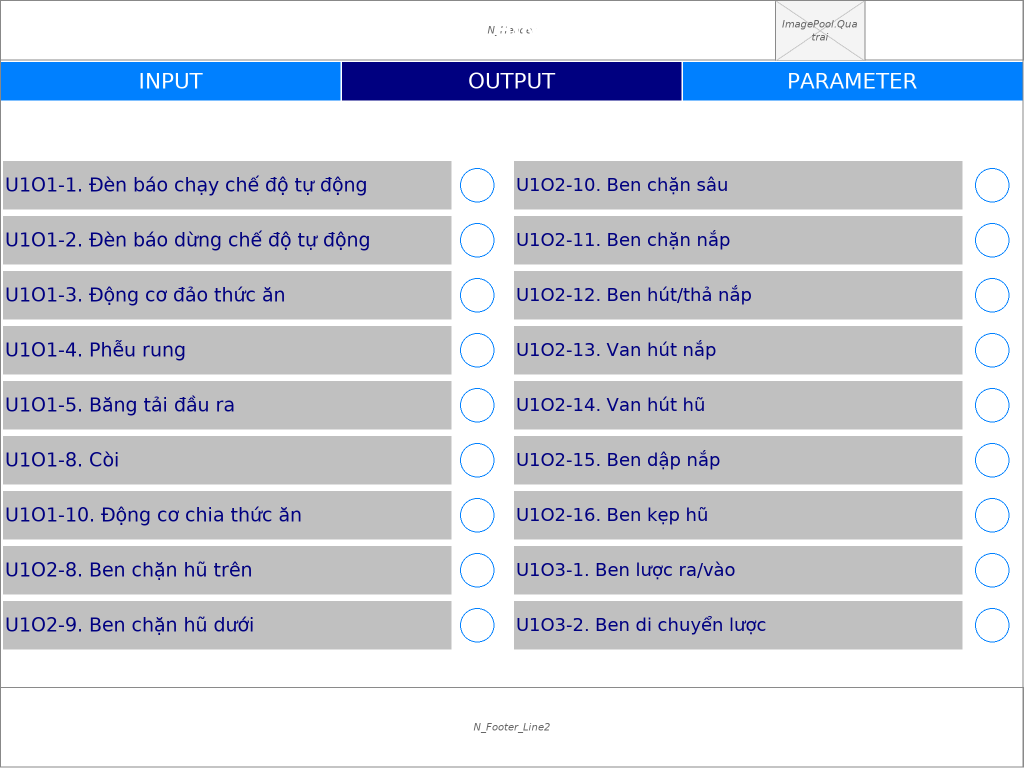
VISUALIZATION N_PLC_O2  // 1024x768
    Frame (0,687 1024x80)
        shows N_Footer_Line2()
    Frame (0,0 1024x60)
        shows N_Header()
    Textfield (353,5 400x50), "MÀN HÌNH IO LINE 2"
    Rectangle (2,160 450x50), "U1O1-1. Đèn báo chạy chế độ tự động"
    Rectangle (2,215 450x50), "U1O1-2. Đèn báo dừng chế độ tự động"
    Rectangle (2,270 450x50), "U1O1-3. Động cơ đảo thức ăn"
    Ellipse (460,168 34x34), colour toggle: GVL_IO.bLight_Running, input disabled if: true
    Ellipse (460,223 34x34), colour toggle: GVL_IO.bLight_Stop, input disabled if: true
    Rectangle (2,325 450x50), "U1O1-4. Phễu rung"
    Rectangle (2,380 450x50), "U1O1-5. Băng tải đầu ra"
    Rectangle (2,435 450x50), "U1O1-8. Còi"
    Rectangle (2,490 450x50), "U1O1-10. Động cơ chia thức ăn"
    Rectangle (2,545 450x50), "U1O2-8. Ben chặn hũ trên"
    Rectangle (2,600 450x50), "U1O2-9. Ben chặn hũ dưới"
    Rectangle (513,160 450x50), "U1O2-10. Ben chặn sâu"
    Rectangle (513,215 450x50), "U1O2-11. Ben chặn nắp"
    Ellipse (460,278 34x34), colour toggle: PR_Line02.fb_FoodMixer.fbInverter.bVFD, input disabled if: true
    Ellipse (460,333 34x34), colour toggle: PR_Line02.fb_WormWeight.fbInverter.bVFD, input disabled if: true
    Ellipse (460,388 34x34), colour toggle: PR_Conveyor_Out.fb_Conveyor.fbInverter.bVFD, input disabled if: true
    Ellipse (460,443 34x34), colour toggle: GVL_IO.bSirens, input disabled if: true
    Ellipse (460,498 34x34), input disabled if: true
    Ellipse (460,553 34x34), colour toggle: PR_Line02.fb_CupSupply.fbCylinder_Up.bMoveExtend, input disabled if: true
    Ellipse (460,608 34x34), colour toggle: PR_Line02.fb_CupSupply.fbCylinder_Dw.bMoveRetract, input disabled if: true
    Ellipse (975,168 34x34), input disabled if: true
    Ellipse (975,223 34x34), colour toggle: PR_Line02.fb_LidSupply.fbCylinder_LidStopper.bMoveRetract, input disabled if: true
    Rectangle (513,270 450x50), "U1O2-12. Ben hút/thả nắp"
    Ellipse (975,278 34x34), input disabled if: true
    Rectangle (513,325 450x50), "U1O2-13. Van hút nắp"
    Rectangle (513,380 450x50), "U1O2-14. Van hút hũ"
    Rectangle (513,435 450x50), "U1O2-15. Ben dập nắp"
    Rectangle (513,490 450x50), "U1O2-16. Ben kẹp hũ"
    Rectangle (513,545 450x50), "U1O3-1. Ben lược ra/vào"
    Rectangle (513,600 450x50), "U1O3-2. Ben di chuyển lược"
    Ellipse (975,333 34x34), input disabled if: true
    Ellipse (975,388 34x34), input disabled if: true
    Ellipse (975,443 34x34), input disabled if: true
    Ellipse (975,498 34x34), colour toggle: PR_Line02.fb_Transfer.fbCylinder_Clip.bMoveRetract, input disabled if: true
    Ellipse (975,553 34x34), colour toggle: PR_Line02.fb_Transfer.fbCylinder_Comb.bMoveExtend, input disabled if: true
    Ellipse (975,608 34x34), colour toggle: PR_Line02.fb_Transfer.fbCylinder_Move_Comb.bMoveExtend, input disabled if: true
    Image (775,0 90x61), image: ImagePool.Qua trai
        OnMouseClick: change screen: N_PLC_O1
    Rectangle (0,61 341x40), "INPUT"
        OnMouseClick: change screen: N_PLC_I2
    Rectangle (341,61 341x40), "OUTPUT"
        OnMouseClick: change screen: N_PLC_O2
    Rectangle (682,61 341x40), "PARAMETER"
        OnMouseClick: change screen: N_Parameter_2
END_VISUALIZATION

(* stored: Version 1.1.0.1, ProductVersion 3.1.4024.12
   Visu N_PLC_O2: Id {f7bf3a36-6474-4c6c-938f-ef48ac59a8cc} *)
